Fanuc KAREL source: kb00181.KL

-- PROVISIONAL review KL for V770-1; original PC SHA256 9707d8f862823b7e0da43d311621a4ae414f6c2ed9e7f2bb822a5fb4088725b7
-- Incomplete behavior may be omitted. Consult companion uncertainty JSON. Do not deploy.
PROGRAM KB00181
%NOLOCKGROUP
BEGIN
  -- UNRESOLVED_PC offsets 5-12; opcodes 9D,23
  -- UNRESOLVED_PC offsets 17-27; opcodes 27,22,31
  -- UNRESOLVED_PC offsets 32-36; opcodes 7F
END KB00181
